SUBAPPLICATION Uebung_010c3_AX (* SoftKey_F1 auf DigitalOutput_Q1 mit GreenWhiteBackground mit Typed Subapp *)
  (* Standard: 61499-2; Description: Copyright (c) 2023 Meisterschulen am Ostbahnhof This program and the accompanying materials are made available under the terms of the Eclipse Public License 2.0 which is available at https://www.eclipse.org/legal/epl-2.0/ SPDX-License-Identifier: EPL-2.0 *)
  (* Version 1.0, 2026-01-15, Franz Höpfinger, Meisterschulen am Ostbahnhof, initial API and implementation and/or initial documentation *)
  PACKAGE Uebungen;
  IMPORT Uebungen::const::UT::DefaultPool::SoftKey_F1;
  IMPORT logiBUS::io::DQ::logiBUS_DO::Output_Q1;
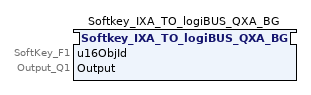
  SUBAPPS
    Softkey_IXA_TO_logiBUS_QXA_BG : MyLib::sys::Softkey_IXA_TO_logiBUS_QXA_BG(u16ObjId := SoftKey_F1, Output := Output_Q1);
  END_SUBAPPS
END_SUBAPPLICATION
